Universal Robots PolyScope program: sequece_testing.urp

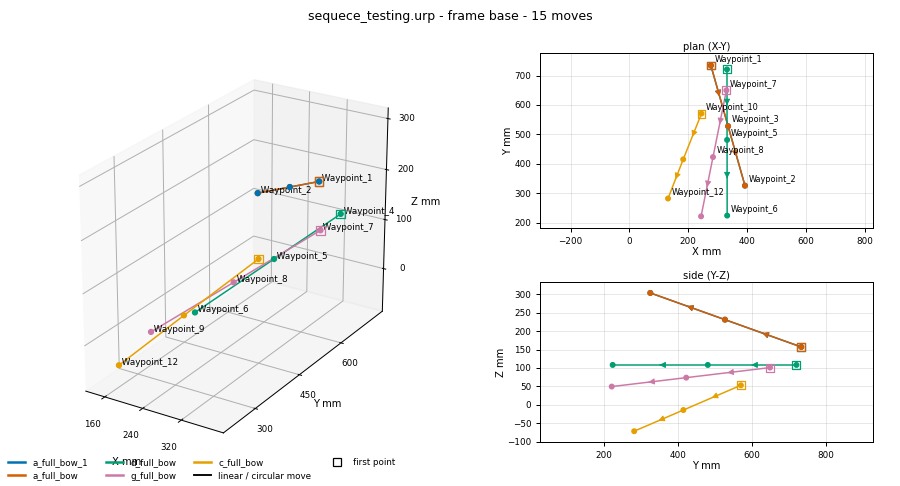
[picture p0: tool path of sequece_testing.urp in frame base, 15 of 18 moves have a stored position in this frame; points joined in program order, loops and branches not executed]
Program sequece_testing (installation=string_planes directory=/programs createdIn=5.17.3 lastSavedIn=5.17.3 robotSerialNumber=20245501435)
Calibrated DH parameters: a=[0.000154, -0.137004, -0.385524, -0.00002, 0.000092, 0]; d=[0.162441, 211.794786, -230.585024, 18.923638, 0.099786, 0.09951]; alpha=[1.569493, -0.001902, 0.003874, 1.570111, -1.570167, 0]; deltaTheta=[0, -1.242934, 1.056292, 0.186646, 0.000002, 0.000001]
InitVariablesNode
Robot Program (runOnlyOnce=true)
  bow_dir := bow_dir≟ True
  note_dir := 1
  Call a_full_bow
  Call a_to_d
  Call d_full_bow
  Call d_to_g
  Call g_full_bow
  Call g_to_c
  Call c_full_bow
SubProgram -> g_to_c
SubProgram -> d_to_g
SubProgram -> a_to_d
SubProgram -> c_full_bow
SubProgram -> g_full_bow
SubProgram -> d_full_bow
SubProgram -> a_full_bow
SubProgram a_full_bow_1 (keepSynchronizedWithDisk=false) programFile=/programs/a_full_bow.urp
  If 
    Placeholder
  MoveL speed 250 mm/s, acceleration 1200 mm/s^2 (useActiveTCP=true) feature=Base
    Waypoint Waypoint_1: TCP in base x=277.237 y=734.032 z=156.892 mm, rx=1.7389 ry=2.3104 rz=-1.1078 rad; joints [-126.647, -28.123, 54.729, -74.616, -91.964, -141.812] deg; TCP offset x=28.21 y=-96.107 z=-99.69 mm, rx=0 ry=0 rz=0 rad
    Waypoint Waypoint_3: motionParameters(blendRadius=0.05); TCP in base x=335.809 y=527.638 z=230.762 mm, rx=1.7389 ry=2.3104 rz=-1.1078 rad; joints [-141.244, -51.172, 87.867, -86.053, -101.589, -152.842] deg
    Waypoint Waypoint_2: TCP in base x=393.128 y=325.659 z=303.053 mm, rx=1.7389 ry=2.3104 rz=-1.1078 rad; joints [-160.523, -67.347, 103.242, -90.17, -113.569, -168.748] deg
SubProgram a_full_bow (keepSynchronizedWithDisk=false) programFile=/programs/a_full_bow.urp
  MoveL speed 250 mm/s, acceleration 1200 mm/s^2 (useActiveTCP=true) feature=Base
    Waypoint Waypoint_1: TCP in base x=277.237 y=734.032 z=156.892 mm, rx=1.7389 ry=2.3104 rz=-1.1078 rad; joints [-126.647, -28.123, 54.729, -74.616, -91.964, -141.812] deg
    Waypoint Waypoint_3: motionParameters(blendRadius=0.05); TCP in base x=335.809 y=527.638 z=230.762 mm, rx=1.7389 ry=2.3104 rz=-1.1078 rad; joints [-141.244, -51.172, 87.867, -86.053, -101.589, -152.842] deg
    Waypoint Waypoint_2: TCP in base x=393.128 y=325.659 z=303.053 mm, rx=1.7389 ry=2.3104 rz=-1.1078 rad; joints [-160.523, -67.347, 103.242, -90.17, -113.569, -168.748] deg
SubProgram a_to_d (keepSynchronizedWithDisk=false) programFile=/programs/a_to_d.urp
  MoveJ speed 60 deg/s, acceleration 80 deg/s^2 (useActiveTCP=true) feature=Base
    Waypoint Waypoint_13 (Relative): relativeFromPosition TCP in base x=343.844 y=499.313 z=240.895 mm, rx=1.7389 ry=2.3104 rz=-1.1077 rad; joints [-143.658, -53.779, 90.874, -86.864, -103.152, -154.726] deg; TCP in base x=332.29 y=455.667 z=108.301 mm, rx=-1.6449 ry=-2.1081 rz=1.059 rad; joints [-146.043, -43.251, 101.393, -102.433, -88.398, -160.538] deg
SubProgram d_full_bow (keepSynchronizedWithDisk=false) programFile=/programs/d_full_bow.urp
  MoveL speed 250 mm/s, acceleration 1200 mm/s^2 (useActiveTCP=true) feature=Base
    Waypoint Waypoint_4: TCP in base x=331.973 y=720.894 z=108.291 mm, rx=-1.645 ry=-2.1081 rz=1.0591 rad; joints [-129.773, -21.651, 52.373, -76.468, -76.907, -149.022] deg
    Waypoint Waypoint_5: motionParameters(blendRadius=0.05); TCP in base x=332.259 y=481.199 z=108.291 mm, rx=-1.645 ry=-2.1081 rz=1.0591 rad; joints [-144.031, -41.816, 97.865, -100.392, -86.961, -159.136] deg
    Waypoint Waypoint_6: TCP in base x=332.566 y=223.853 z=108.291 mm, rx=-1.645 ry=-2.1081 rz=1.0591 rad; joints [-170.229, -51.627, 126.122, -120.942, -105.516, -177.767] deg
SubProgram d_to_g (keepSynchronizedWithDisk=false) programFile=/programs/d_to_g.urp
  MoveJ speed 60 deg/s, acceleration 80 deg/s^2 (useActiveTCP=true) feature=Base
    Waypoint Waypoint_14 (Relative): relativeFromPosition TCP in base x=332.29 y=455.66 z=108.297 mm, rx=-1.6449 ry=-2.1081 rz=1.0591 rad; joints [-146.043, -43.251, 101.394, -102.431, -88.399, -160.539] deg; TCP in base x=285.729 y=429.531 z=74.701 mm, rx=-1.7275 ry=-1.8378 rz=0.7436 rad; joints [-145.706, -41.272, 112.343, -121.516, -69.317, -156.458] deg
SubProgram g_full_bow (keepSynchronizedWithDisk=false) programFile=/programs/g_full_bow.urp
  MoveL speed 250 mm/s, acceleration 1200 mm/s^2 (useActiveTCP=true) feature=Base
    Waypoint Waypoint_7: TCP in base x=329.981 y=649.486 z=101.065 mm, rx=-1.7033 ry=-1.7268 rz=0.636 rad; joints [-132.743, -28.556, 74.955, -104.888, -53.814, -143.829] deg
    Waypoint Waypoint_8: motionParameters(blendRadius=0.05); TCP in base x=284.388 y=422.807 z=73.9 mm, rx=-1.7281 ry=-1.8411 rz=0.747 rad; joints [-146.247, -41.489, 113.29, -122.055, -69.91, -156.899] deg
    Waypoint Waypoint_9: TCP in base x=243.857 y=221.298 z=49.751 mm, rx=-1.7452 ry=-1.9422 rz=0.8491 rad; joints [-169.181, -41.825, 137.541, -143.377, -92.671, -173.897] deg
SubProgram g_to_c (keepSynchronizedWithDisk=false) programFile=/programs/g_to_c.urp
  MoveJ speed 60 deg/s, acceleration 80 deg/s^2 (useActiveTCP=true) feature=Base
    Waypoint Waypoint_15 (Relative): relativeFromPosition TCP in base x=285.259 y=429.339 z=74.177 mm, rx=-1.7286 ry=-1.8348 rz=0.7402 rad; joints [-145.697, -41.207, 112.434, -121.773, -69.122, -156.372] deg; TCP in base x=183.045 y=414.877 z=-13.795 mm, rx=-1.8417 ry=-1.5193 rz=0.1582 rad; joints [-140.01, -22.062, 119.511, -179.217, -47.149, -131.928] deg
SubProgram c_full_bow (keepSynchronizedWithDisk=false) programFile=/programs/c_full_bow.urp
  MoveL speed 250 mm/s, acceleration 1200 mm/s^2 (useActiveTCP=true) feature=Base
    Waypoint Waypoint_10: TCP in base x=245.284 y=570.71 z=53.266 mm, rx=-1.8425 ry=-1.3918 rz=0.0687 rad; joints [-132.226, -24.798, 96.314, -169.322, -42.692, -112.607] deg
    Waypoint Waypoint_11: TCP in base x=183.128 y=415.066 z=-13.712 mm, rx=-1.8418 ry=-1.5191 rz=0.1581 rad; joints [-139.998, -22.072, 119.488, -179.203, -47.14, -131.9] deg
    Waypoint Waypoint_12: TCP in base x=131.526 y=281.987 z=-70.972 mm, rx=-1.836 ry=-1.6275 rz=0.2368 rad; joints [-152.883, -9.471, 132.363, -190.356, -55.903, -152.614] deg
